FUNCTION_BLOCK GF_Halten EXTENDS FB_Basisfunktionalitaeten
VAR_INPUT
	// Instanzieren von Sensoren mit Interfaces
	
	// Instanzieren von Aktoren mit Interfaces
	
END_VAR
VAR_OUTPUT
	
END_VAR
VAR
	
END_VAR

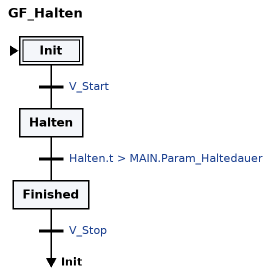
INITIAL_STEP Init:
END_STEP
TRANSITION FROM Init TO Halten
    := V_Start;
END_TRANSITION
STEP Halten:
END_STEP
TRANSITION FROM Halten TO Finished
    := Halten.t > MAIN.Param_Haltedauer;
END_TRANSITION
STEP Finished:
END_STEP
TRANSITION FROM Finished TO Init
    := V_Stop;
END_TRANSITION

END_FUNCTION_BLOCK

(* stored: Version 1.1.0.1, ProductVersion 3.1.4024.12
   POU GF_Halten: Id {d2875f49-552d-4f37-905a-2f2ecd102667}, SpecialFunc None *)
